PROGRAM MAIN
VAR
	LS_Floor:ARRAY[1..3]	OF	ST_LevelSensors;
	BT_FloorCall AT %I*:ARRAY[1..3]	OF	BOOL;
	Elevator:FB_Motor;
	STATE: E_States;
	RequestedFloor: INT;
	i: INT;
	CurrentFloor: INT;
	PulseTrigger:ARRAY[1..3]OF	TP;
	LatchTime: ULINT;
	ElapsedTime: LTIME;
END_VAR


CASE STATE	OF	
	E_States.Call:;
		//action logic
		FOR	i:=1 TO 3	DO
			IF	BT_FloorCall[i]	THEN
				RequestedFloor:=i;
				LatchTime:=F_GetSystemTime();
				EXIT;
			END_IF
		END_FOR
		//transitions
		IF	RequestedFloor>CurrentFloor	THEN
			STATE:=E_States.MoveUp;
		ELSIF	RequestedFloor<CurrentFloor	THEN
			STATE:=E_States.MoveDown;
		END_IF
		
		//initialise pulse timer
		FOR	i:=1	TO	3	DO
			PulseTrigger[i](IN:=FALSE);
		END_FOR
		
	E_States.MoveUp:
		Elevator.MoveUp();
		FOR	i:=1	TO	3	DO
			PulseTrigger[i](IN:=LS_Floor[i].Low,PT:=T#10MS);
			IF	PulseTrigger[i].Q	THEN
				STATE:=E_States.IncrementFloor;
			END_IF
		END_FOR
		IF	RequestedFloor=CurrentFloor	THEN	
			state:=E_States.SlowDown;
		END_IF
		
	E_States.MoveDown:
		Elevator.MoveDown();
		FOR	i:=1	TO	3	DO
			PulseTrigger[i](IN:=LS_Floor[i].High,PT:=T#10MS);
			IF	PulseTrigger[i].Q	THEN
				STATE:=E_States.DecrementFloor;
			END_IF
		END_FOR
		IF	RequestedFloor=CurrentFloor	THEN	
			state:=E_States.SlowDown;
		END_IF
		
	E_States.IncrementFloor:
		CurrentFloor:=CurrentFloor+1;
		STATE:=E_States.MoveUp;
	E_States.DecrementFloor:
		CurrentFloor:=CurrentFloor-1;
		STATE:=E_States.MoveDown;
	E_States.SlowDown:
		Elevator.SlowDown();
		FOR	i:=1	TO	3	DO
			IF	LS_Floor[i].Mid	THEN
				STATE:=E_States.Stop;
			END_IF
		END_FOR
	E_States.Stop:
		//ElapsedTime:=ULINT_TO_LTIME(F_GetSystemTime()-LatchTime);
		Elevator.Stop();
		state:=E_States.Call;
END_CASE

END_PROGRAM

(* stored: Version 1.1.0.1, ProductVersion 3.1.4024.11
   POU MAIN: Id {fd6255af-2d3d-47fe-bc9f-2b7654d26df2}, SpecialFunc None *)
